// TIA Portal V17 export
// export: Created 2022-07-28T18:03:03.4522009Z, ExportSetting None, DisplayName Totally Integrated Automation Portal, DisplayVersion V17, DisplayName TIA Portal Openness, DisplayVersion V17, DisplayName TIA Portal Teamcenter Gateway, DisplayVersion V17, DisplayName TIA Portal Version Control Interface, DisplayVersion V17, DisplayName TIA Portal Test Suite Advanced, DisplayVersion V17, DisplayName SINAMICS Startdrive Advanced, DisplayVersion V17, DisplayName SINAMICS DCC, DisplayVersion V17, DisplayName SINAMICS Startdrive G130, G150, S120, S150, SINAMICS MV, S210, DisplayVersion V17, DisplayName SINAMICS Startdrive G110M, G120, G120C, G120D, G120P, G115D, DisplayVersion V17, DisplayName STEP 7 Professional, DisplayVersion V17, DisplayName SIMATIC Energy Suite, DisplayVersion V17, DisplayName STEP 7 CFC, DisplayVersion V17, DisplayName STEP 7 Safety, DisplayVersion V17, DisplayName WinCC Advanced / Unified PC, DisplayVersion V17, DisplayName SIMATIC Visualization Architect, DisplayVersion V17
DATA_BLOCK "D_PLC_CycleInfo_DATA"   // DB6
{ S7_Optimized_Access := 'TRUE' }
// stored: MemoryReserve 100
   VAR RETAIN
      Config : Struct
         Max_Number_Groups { S7_SetPoint := 'True'} : Int := 3;
         Max_Number_ButtonInGroup : Int := 5;
      END_STRUCT;
   END_VAR
   VAR
      Grp_Obj { ExternalAccessible := 'False'; ExternalVisible := 'False'; ExternalWritable := 'False'} : Array[0..9, 0..15] of "Lib_PLC_CycleInfo";
      "Grp_HMI&CNTR" : Array[0..9, 0..15] of "Lib_PLC_CycleInfo";
   END_VAR
BEGIN
   // Grp_Obj[0,0] : Система в цілому
   // "Grp_HMI&CNTR"[0,0] : Система - сумарно
   // "Grp_HMI&CNTR"[0,1] : not used
   // "Grp_HMI&CNTR"[0,2] : not used
   // "Grp_HMI&CNTR"[0,3] : not used
   // "Grp_HMI&CNTR"[0,4] : not used
   // "Grp_HMI&CNTR"[0,5] : not used
   // "Grp_HMI&CNTR"[0,6] : not used
   // "Grp_HMI&CNTR"[0,7] : not used
   // "Grp_HMI&CNTR"[0,8] : not used
   // "Grp_HMI&CNTR"[0,9] : not used
   // "Grp_HMI&CNTR"[0,10] : not used
   // "Grp_HMI&CNTR"[0,11] : not used
   // "Grp_HMI&CNTR"[0,12] : not used
   // "Grp_HMI&CNTR"[0,13] : not used
   // "Grp_HMI&CNTR"[0,14] : not used
   // "Grp_HMI&CNTR"[0,15] : not used
   // "Grp_HMI&CNTR"[1,0] : Група 1 - сумарно
   // "Grp_HMI&CNTR"[1,1] : Група 1 - Підгрупа 1
   // "Grp_HMI&CNTR"[1,2] : Група 1 - Підгрупа 2
   // "Grp_HMI&CNTR"[1,3] : Група 1 - Підгрупа 3
   // "Grp_HMI&CNTR"[1,4] : Група 1 - Підгрупа 4
   // "Grp_HMI&CNTR"[1,5] : Група 1 - Підгрупа 5
   // "Grp_HMI&CNTR"[1,6] : Група 1 - Підгрупа 6
   // "Grp_HMI&CNTR"[1,7] : Група 1 - Підгрупа 7
   // "Grp_HMI&CNTR"[1,8] : Група 1 - Підгрупа 8
   // "Grp_HMI&CNTR"[1,9] : Група 1 - Підгрупа 9
   // "Grp_HMI&CNTR"[1,10] : Група 1 - Підгрупа 10
   // "Grp_HMI&CNTR"[1,11] : Група 1 - Підгрупа 11
   // "Grp_HMI&CNTR"[1,12] : Група 1 - Підгрупа 12
   // "Grp_HMI&CNTR"[1,13] : Група 1 - Підгрупа 13
   // "Grp_HMI&CNTR"[1,14] : Група 1 - Підгрупа 14
   // "Grp_HMI&CNTR"[1,15] : Група 1 - Підгрупа 15
   // "Grp_HMI&CNTR"[2,0] : Група 2 - сумарно
   // "Grp_HMI&CNTR"[2,1] : Група 2 - Підгрупа 1
   // "Grp_HMI&CNTR"[2,2] : Група 2 - Підгрупа 2
   // "Grp_HMI&CNTR"[2,3] : Група 2 - Підгрупа 3
   // "Grp_HMI&CNTR"[2,4] : Група 2 - Підгрупа 4
   // "Grp_HMI&CNTR"[2,5] : Група 2 - Підгрупа 5
   // "Grp_HMI&CNTR"[2,6] : Група 2 - Підгрупа 6
   // "Grp_HMI&CNTR"[2,7] : Група 2 - Підгрупа 7
   // "Grp_HMI&CNTR"[2,8] : Група 2 - Підгрупа 8
   // "Grp_HMI&CNTR"[2,9] : Група 2 - Підгрупа 9
   // "Grp_HMI&CNTR"[2,10] : Група 2 - Підгрупа 10
   // "Grp_HMI&CNTR"[2,11] : Група 2 - Підгрупа 11
   // "Grp_HMI&CNTR"[2,12] : Група 2 - Підгрупа 12
   // "Grp_HMI&CNTR"[2,13] : Група 2 - Підгрупа 13
   // "Grp_HMI&CNTR"[2,14] : Група 2 - Підгрупа 14
   // "Grp_HMI&CNTR"[2,15] : Група 2 - Підгрупа 15
   // "Grp_HMI&CNTR"[3,0] : Група 3 - сумарно
   // "Grp_HMI&CNTR"[3,1] : Група 3 - Підгрупа 1
   // "Grp_HMI&CNTR"[3,2] : Група 3 - Підгрупа 2
   // "Grp_HMI&CNTR"[3,3] : Група 3 - Підгрупа 3
   // "Grp_HMI&CNTR"[3,4] : Група 3 - Підгрупа 4
   // "Grp_HMI&CNTR"[3,5] : Група 3 - Підгрупа 5
   // "Grp_HMI&CNTR"[3,6] : Група 3 - Підгрупа 6
   // "Grp_HMI&CNTR"[3,7] : Група 3 - Підгрупа 7
   // "Grp_HMI&CNTR"[3,8] : Група 3 - Підгрупа 8
   // "Grp_HMI&CNTR"[3,9] : Група 3 - Підгрупа 9
   // "Grp_HMI&CNTR"[3,10] : Група 3 - Підгрупа 10
   // "Grp_HMI&CNTR"[3,11] : Група 3 - Підгрупа 11
   // "Grp_HMI&CNTR"[3,12] : Група 3 - Підгрупа 12
   // "Grp_HMI&CNTR"[3,13] : Група 3 - Підгрупа 13
   // "Grp_HMI&CNTR"[3,14] : Група 3 - Підгрупа 14
   // "Grp_HMI&CNTR"[3,15] : Група 3 - Підгрупа 15
   // "Grp_HMI&CNTR"[4,0] : Група 4 - сумарно
   // "Grp_HMI&CNTR"[4,1] : Група 4 - Підгрупа 1
   // "Grp_HMI&CNTR"[4,2] : Група 4 - Підгрупа 2
   // "Grp_HMI&CNTR"[4,3] : Група 4 - Підгрупа 3
   // "Grp_HMI&CNTR"[4,4] : Група 4 - Підгрупа 4
   // "Grp_HMI&CNTR"[4,5] : Група 4 - Підгрупа 5
   // "Grp_HMI&CNTR"[4,6] : Група 4 - Підгрупа 6
   // "Grp_HMI&CNTR"[4,7] : Група 4 - Підгрупа 7
   // "Grp_HMI&CNTR"[4,8] : Група 4 - Підгрупа 8
   // "Grp_HMI&CNTR"[4,9] : Група 4 - Підгрупа 9
   // "Grp_HMI&CNTR"[4,10] : Група 4 - Підгрупа 10
   // "Grp_HMI&CNTR"[4,11] : Група 4 - Підгрупа 11
   // "Grp_HMI&CNTR"[4,12] : Група 4 - Підгрупа 12
   // "Grp_HMI&CNTR"[4,13] : Група 4 - Підгрупа 13
   // "Grp_HMI&CNTR"[4,14] : Група 4 - Підгрупа 14
   // "Grp_HMI&CNTR"[4,15] : Група 4 - Підгрупа 15
   // "Grp_HMI&CNTR"[5,0] : Група 5 - сумарно
   // "Grp_HMI&CNTR"[5,1] : Група 5 - Підгрупа 1
   // "Grp_HMI&CNTR"[5,2] : Група 5 - Підгрупа 2
   // "Grp_HMI&CNTR"[5,3] : Група 5 - Підгрупа 3
   // "Grp_HMI&CNTR"[5,4] : Група 5 - Підгрупа 4
   // "Grp_HMI&CNTR"[5,5] : Група 5 - Підгрупа 5
   // "Grp_HMI&CNTR"[5,6] : Група 5 - Підгрупа 6
   // "Grp_HMI&CNTR"[5,7] : Група 5 - Підгрупа 7
   // "Grp_HMI&CNTR"[5,8] : Група 5 - Підгрупа 8
   // "Grp_HMI&CNTR"[5,9] : Група 5 - Підгрупа 9
   // "Grp_HMI&CNTR"[5,10] : Група 5 - Підгрупа 10
   // "Grp_HMI&CNTR"[5,11] : Група 5 - Підгрупа 11
   // "Grp_HMI&CNTR"[5,12] : Група 5 - Підгрупа 12
   // "Grp_HMI&CNTR"[5,13] : Група 5 - Підгрупа 13
   // "Grp_HMI&CNTR"[5,14] : Група 5 - Підгрупа 14
   // "Grp_HMI&CNTR"[5,15] : Група 5 - Підгрупа 15
   // "Grp_HMI&CNTR"[6,0] : Група 6 - сумарно
   // "Grp_HMI&CNTR"[6,1] : Група 6 - Підгрупа 1
   // "Grp_HMI&CNTR"[6,2] : Група 6 - Підгрупа 2
   // "Grp_HMI&CNTR"[6,3] : Група 6 - Підгрупа 3
   // "Grp_HMI&CNTR"[6,4] : Група 6 - Підгрупа 4
   // "Grp_HMI&CNTR"[6,5] : Група 6 - Підгрупа 5
   // "Grp_HMI&CNTR"[6,6] : Група 6 - Підгрупа 6
   // "Grp_HMI&CNTR"[6,7] : Група 6 - Підгрупа 7
   // "Grp_HMI&CNTR"[6,8] : Група 6 - Підгрупа 8
   // "Grp_HMI&CNTR"[6,9] : Група 6 - Підгрупа 9
   // "Grp_HMI&CNTR"[6,10] : Група 6 - Підгрупа 10
   // "Grp_HMI&CNTR"[6,11] : Група 6 - Підгрупа 11
   // "Grp_HMI&CNTR"[6,12] : Група 6 - Підгрупа 12
   // "Grp_HMI&CNTR"[6,13] : Група 6 - Підгрупа 13
   // "Grp_HMI&CNTR"[6,14] : Група 6 - Підгрупа 14
   // "Grp_HMI&CNTR"[6,15] : Група 6 - Підгрупа 15
   // "Grp_HMI&CNTR"[7,0] : Група 7 - сумарно
   // "Grp_HMI&CNTR"[7,1] : Група 7 - Підгрупа 1
   // "Grp_HMI&CNTR"[7,2] : Група 7 - Підгрупа 2
   // "Grp_HMI&CNTR"[7,3] : Група 7 - Підгрупа 3
   // "Grp_HMI&CNTR"[7,4] : Група 7 - Підгрупа 4
   // "Grp_HMI&CNTR"[7,5] : Група 7 - Підгрупа 5
   // "Grp_HMI&CNTR"[7,6] : Група 7 - Підгрупа 6
   // "Grp_HMI&CNTR"[7,7] : Група 7 - Підгрупа 7
   // "Grp_HMI&CNTR"[7,8] : Група 7 - Підгрупа 8
   // "Grp_HMI&CNTR"[7,9] : Група 7 - Підгрупа 9
   // "Grp_HMI&CNTR"[7,10] : Група 7 - Підгрупа 10
   // "Grp_HMI&CNTR"[7,11] : Група 7 - Підгрупа 11
   // "Grp_HMI&CNTR"[7,12] : Група 7 - Підгрупа 12
   // "Grp_HMI&CNTR"[7,13] : Група 7 - Підгрупа 13
   // "Grp_HMI&CNTR"[7,14] : Група 7 - Підгрупа 14
   // "Grp_HMI&CNTR"[7,15] : Група 7 - Підгрупа 15
   // "Grp_HMI&CNTR"[8,0] : Група 8 - сумарно
   // "Grp_HMI&CNTR"[8,1] : Група 8 - Підгрупа 1
   // "Grp_HMI&CNTR"[8,2] : Група 8 - Підгрупа 2
   // "Grp_HMI&CNTR"[8,3] : Група 8 - Підгрупа 3
   // "Grp_HMI&CNTR"[8,4] : Група 8 - Підгрупа 4
   // "Grp_HMI&CNTR"[8,5] : Група 8 - Підгрупа 5
   // "Grp_HMI&CNTR"[8,6] : Група 8 - Підгрупа 6
   // "Grp_HMI&CNTR"[8,7] : Група 8 - Підгрупа 7
   // "Grp_HMI&CNTR"[8,8] : Група 8 - Підгрупа 8
   // "Grp_HMI&CNTR"[8,9] : Група 8 - Підгрупа 9
   // "Grp_HMI&CNTR"[8,10] : Група 8 - Підгрупа 10
   // "Grp_HMI&CNTR"[8,11] : Група 8 - Підгрупа 11
   // "Grp_HMI&CNTR"[8,12] : Група 8 - Підгрупа 12
   // "Grp_HMI&CNTR"[8,13] : Група 8 - Підгрупа 13
   // "Grp_HMI&CNTR"[8,14] : Група 8 - Підгрупа 14
   // "Grp_HMI&CNTR"[8,15] : Група 8 - Підгрупа 15
   // "Grp_HMI&CNTR"[9,0] : Група 9 - сумарно
   // "Grp_HMI&CNTR"[9,1] : Група 9 - Підгрупа 1
   // "Grp_HMI&CNTR"[9,2] : Група 9 - Підгрупа 2
   // "Grp_HMI&CNTR"[9,3] : Група 9 - Підгрупа 3
   // "Grp_HMI&CNTR"[9,4] : Група 9 - Підгрупа 4
   // "Grp_HMI&CNTR"[9,5] : Група 9 - Підгрупа 5
   // "Grp_HMI&CNTR"[9,6] : Група 9 - Підгрупа 6
   // "Grp_HMI&CNTR"[9,7] : Група 9 - Підгрупа 7
   // "Grp_HMI&CNTR"[9,8] : Група 9 - Підгрупа 8
   // "Grp_HMI&CNTR"[9,9] : Група 9 - Підгрупа 9
   // "Grp_HMI&CNTR"[9,10] : Група 9 - Підгрупа 10
   // "Grp_HMI&CNTR"[9,11] : Група 9 - Підгрупа 11
   // "Grp_HMI&CNTR"[9,12] : Група 9 - Підгрупа 12
   // "Grp_HMI&CNTR"[9,13] : Група 9 - Підгрупа 13
   // "Grp_HMI&CNTR"[9,14] : Група 9 - Підгрупа 14
   // "Grp_HMI&CNTR"[9,15] : Група 9 - Підгрупа 15
END_DATA_BLOCK
